RoboDK station: ejercicioRobotCilindro.rdk

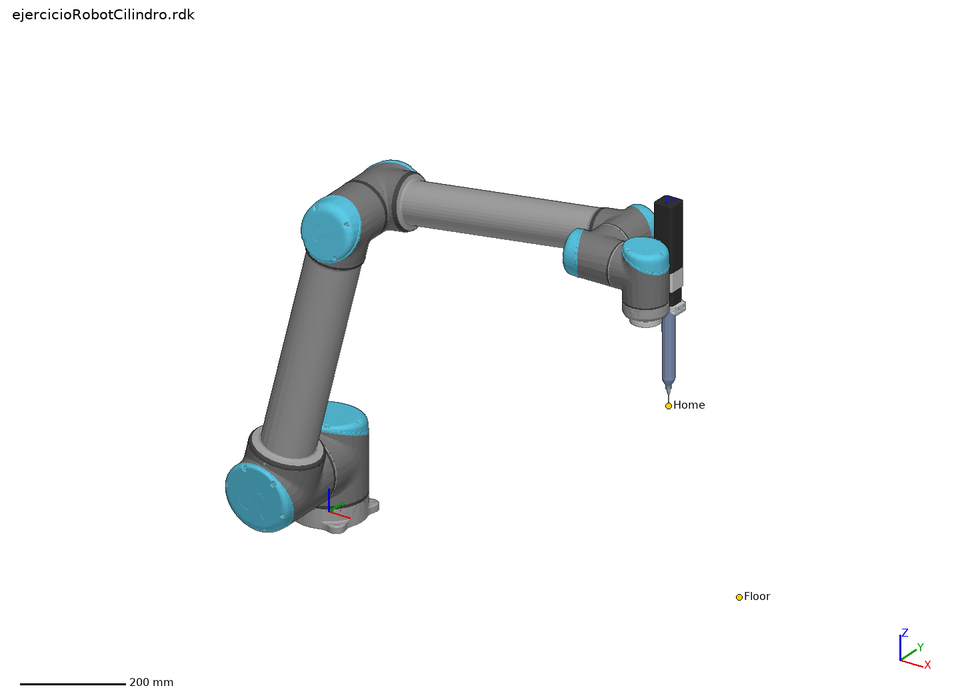
[picture v0: the station drawn from its stored meshes, robots at their saved joint values, targets as dots, program paths as lines]
Station tarea 4 completa (saved by RoboDK 6.0.4). Poses are relative to the parent item; angles as X-Y-Z fixed-axis rotations.
  - frame UR10 Base at (2.24, 45.03, 606.3) mm
    - robot UR10: 6 axes, payload 10 kg, reach 1300 mm, repeatability 0.1 mm, weight 28.9 kg
        modified DH rows (alpha deg, a mm, theta deg, d mm): 0, 0, 0, 128; 90, 0, 180, 0; 0, 612.7, 0, 0; 0, 571.6, 0, 163.9; -90, 0, 0, 115.7; 90, 0, 180, 92.2
        joint limits [-360, -360, -360, -360, -360, -360] to [360, 360, 360, 360, 360, 360]; home [0, -90, -90, 0, 90, 0]; saved at [1.302, -103.964, -68.526, -97.51, 90, -88.698]
      - tool Dispenser , TCP at (0, -75, 221.24) mm, rotated rx 0 ry 0 rz 90 deg, size 63 x 128.2 x 432.2 mm
    - target Home (Cartesian target) at (833.75, -70, 483.87) mm, rotated rx 180 ry 0 rz -90 deg; joints [1.302, -103.964, -68.526, -97.51, 90, -88.698] of UR10
    - target Floor (Cartesian target) at (892.49, 80, 37.72) mm, rotated rx -179.06 ry 0 rz -90 deg; joints [10.966, -117.608, -96.64, -54.833, 89.822, -79.035] of UR10
  - Python program Cilindro (listed below)
  - Python program cono invertido (listed below)
  - Python program Cono positivo (listed below)

--- Python program Cilindro ---
# Importamos Librerias
from robodk.robolink import *
from robodk.robomath import *

#Crear Instancia de la Clase RoboLink
rLink = Robolink()

#Obtenemos el Robot selecionado
Robot = rLink.Item('',ITEM_TYPE_ROBOT)

#Vincular variables de Python con targets
varHome = rLink.Item('Home')
varSuelo = rLink.Item('Floor')


# Comprovar el movimiento del robot.
Robot.MoveL(varHome)
Robot.MoveL(varSuelo)

#Obtener la Posicion de Referencia (Pose)
PosRef = varSuelo.Pose()
PosRefAltura = varHome.Pose()

#Pedirle al Usuario Ingrese Vertices.
#Vertices = int(mbox('Ingrese Numero de Vertices: ',entry=True))
Vertices = 360

# Crear Forma Geometria en el Plano.
for i in range(Vertices + 1):
    Angulo = i * 2 * pi / (Vertices)     #Convierte a grados
    Posei = PosRef * rotz(Angulo) * transl(100,0,0) * rotz(-Angulo)
    PoseiAlt= PosRefAltura*rotz(Angulo)*transl(100,0,0)*rotz(-Angulo)
    # Pasar como parametro al movimiento del Robot
    Robot.MoveL(Posei)

    #Proyecta Linea al plano alterno (Altura)
    Robot.MoveL(PoseiAlt)

    # Regresa al Plano Original (Suelo)
    Robot.MoveL(Posei)

Eje_Z = 0
# Crear Forma Geometria en el Plano.
for i in range (50):
    for i in range(Vertices + 1):
        Angulo = i * 2 * pi / (Vertices)     #Convierte a grados
        Posei = PosRef * rotz(Angulo) * transl(100,0,Eje_Z) * rotz(-Angulo)
        Eje_Z = Eje_Z - 0.01

        # Dibuja la trayectoria mediante el movimiento del Robot
        Robot.MoveL(Posei)
Robot.MoveL(varHome)

--- Python program cono invertido ---
from robodk.robolink import *
from robodk.robomath import *

# ----------------------------------
# Conexión con RoboDK
# ----------------------------------
RDK = Robolink()

# Seleccionar robot
Robot = RDK.Item('', ITEM_TYPE_ROBOT)

if not Robot.Valid():
    raise Exception('No se encontró ningún robot.')

# Targets de referencia
Home = RDK.Item('Home')
Floor = RDK.Item('Floor')

if not Home.Valid():
    raise Exception('No existe el target Home.')

if not Floor.Valid():
    raise Exception('No existe el target Floor.')

# ----------------------------------
# Movimiento inicial
# ----------------------------------
Robot.MoveL(Home)
Robot.MoveL(Floor)

# Pose de referencia
PosRef = Floor.Pose()

# ----------------------------------
# Parámetros del cono
# ----------------------------------
RadioBase = 100.0      # mm
AlturaCono = 200.0     # mm

Capas = 100            # Cantidad de niveles del cono
Vertices = 360         # Resolución de cada circunferencia

# ----------------------------------
# Dibujo del cono
# ----------------------------------
for capa in range(Capas + 1):

    # Altura actual
    Zactual = AlturaCono * capa / Capas

    # Radio decreciente
    RadioActual = RadioBase * (1 - capa / Capas)

    # Dibujar circunferencia
    for punto in range(Vertices + 1):

        Angulo = punto * 2 * pi / Vertices

        Posei = PosRef * \
                rotz(Angulo) * \
                transl(RadioActual, 0, Zactual) * \
                rotz(-Angulo)

        Robot.MoveL(Posei)

# ----------------------------------
# Llegar exactamente al vértice
# ----------------------------------
PoseVertice = PosRef * transl(0, 0, AlturaCono)
Robot.MoveL(PoseVertice)

# ----------------------------------
# Regresar a Home
# ----------------------------------
Robot.MoveL(Home)

--- Python program Cono positivo ---
from robodk.robolink import *
from robodk.robomath import *

RDK = Robolink()
Robot = RDK.Item('', ITEM_TYPE_ROBOT)

Home = RDK.Item('Home')
Floor = RDK.Item('Floor')

Robot.MoveL(Home)
Robot.MoveL(Floor)

PosRef = Floor.Pose()

RadioBase = 100.0
AlturaCono = 200.0

Capas = 60        #  reducido para estabilidad
Vertices = 120    #  reducido para evitar errores

# ----------------------------------
# DIBUJO DEL CONO
# ----------------------------------
for capa in range(Capas + 1):

    Zactual = -AlturaCono * capa / Capas
    RadioActual = RadioBase * (1 - capa / Capas)

    for punto in range(Vertices + 1):

        ang = 2 * pi * punto / Vertices

        x = RadioActual * cos(ang)
        y = RadioActual * sin(ang)

        Posei = PosRef * transl(x, y, Zactual)

        #  SOLO MOVER SI ES ALCANZABLE
        if Robot.SolveIK(Posei).list():

            try:
                Robot.MoveL(Posei)
            except:
                pass

# ----------------------------------
# VÉRTICE FINAL
# ----------------------------------
PoseVertice = PosRef * transl(0, 0, -AlturaCono)

if Robot.SolveIK(PoseVertice).list():
    Robot.MoveL(PoseVertice)

Robot.MoveL(Home)
